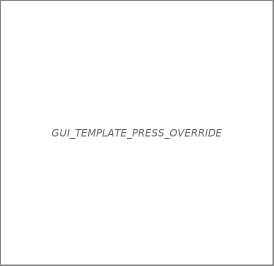
VISUALIZATION GUI_P2_OVERRIDE  // 274x266
    Frame (0,0 274x266)
        shows GUI_TEMPLATE_PRESS_OVERRIDE(m_Cmd := MAIN.pressOR_P1, m_Press := MAIN.P1)
END_VISUALIZATION

(* stored: Version 1.1.0.1, ProductVersion 3.1.4024.12
   Visu GUI_P2_OVERRIDE: Id {7e0cbadd-d964-46f4-8c95-a05ff3b36add} *)
